SUBAPPLICATION Uebung_006_SAFE_AX_02 (* Wie Uebung_006_SAFE_AX, aber mit SF_EmergencyStop statt StartPermit/StartGate *)
  (* Standard: 61499-2; Description: Copyright (c) 2026 Meisterschulen am Ostbahnhof This program and the accompanying materials are made available under the terms of the Eclipse Public License 2.0 which is available at https://www.eclipse.org/legal/epl-2.0/ SPDX-License-Identifier: EPL-2.0 *)
  (* Version 1.0, 2026-10-09, Franz Höpfinger, Meisterschulen am Ostbahnhof, Zweite SAFE-Variante von Uebung_006_AX, diesmal mit dem PLCopen-Standardbaustein SF_EmergencyStop (Part 1 Ch. 6.5) statt der handgebauten StartPermit(E_RS)/StartGate(E_PERMIT)-Loesung aus Uebung_006_SAFE_AX. SF_EmergencyStop und SF_ResetButton sind im eingebetteten Muster (Figure 13 der Spec) ueber ResetRequest/ResetRequested verkoppelt: EmergencyStop fordert ResetButton nur dann zur Ueberwachung an, wenn tatsaechlich ein Reset noetig ist. S_StartReset=FALSE und S_AutoReset=FALSE: kein automatischer Wiederanlauf, RESET (I7) ist immer zwingend erforderlich. *)
  PACKAGE Uebungen;
  IMPORT logiBUS::io::DI::logiBUS_DI::Input_I1;
  IMPORT logiBUS::io::DI::logiBUS_DI::Input_I2;
  IMPORT logiBUS::io::DI::logiBUS_DI::Input_I7;
  IMPORT logiBUS::io::DI::logiBUS_DI::Input_I8;
  IMPORT logiBUS::io::DI::logiBUS_DI_Events::BUTTON_SINGLE_CLICK;
  IMPORT logiBUS::io::DQ::logiBUS_DO::Output_Q1;
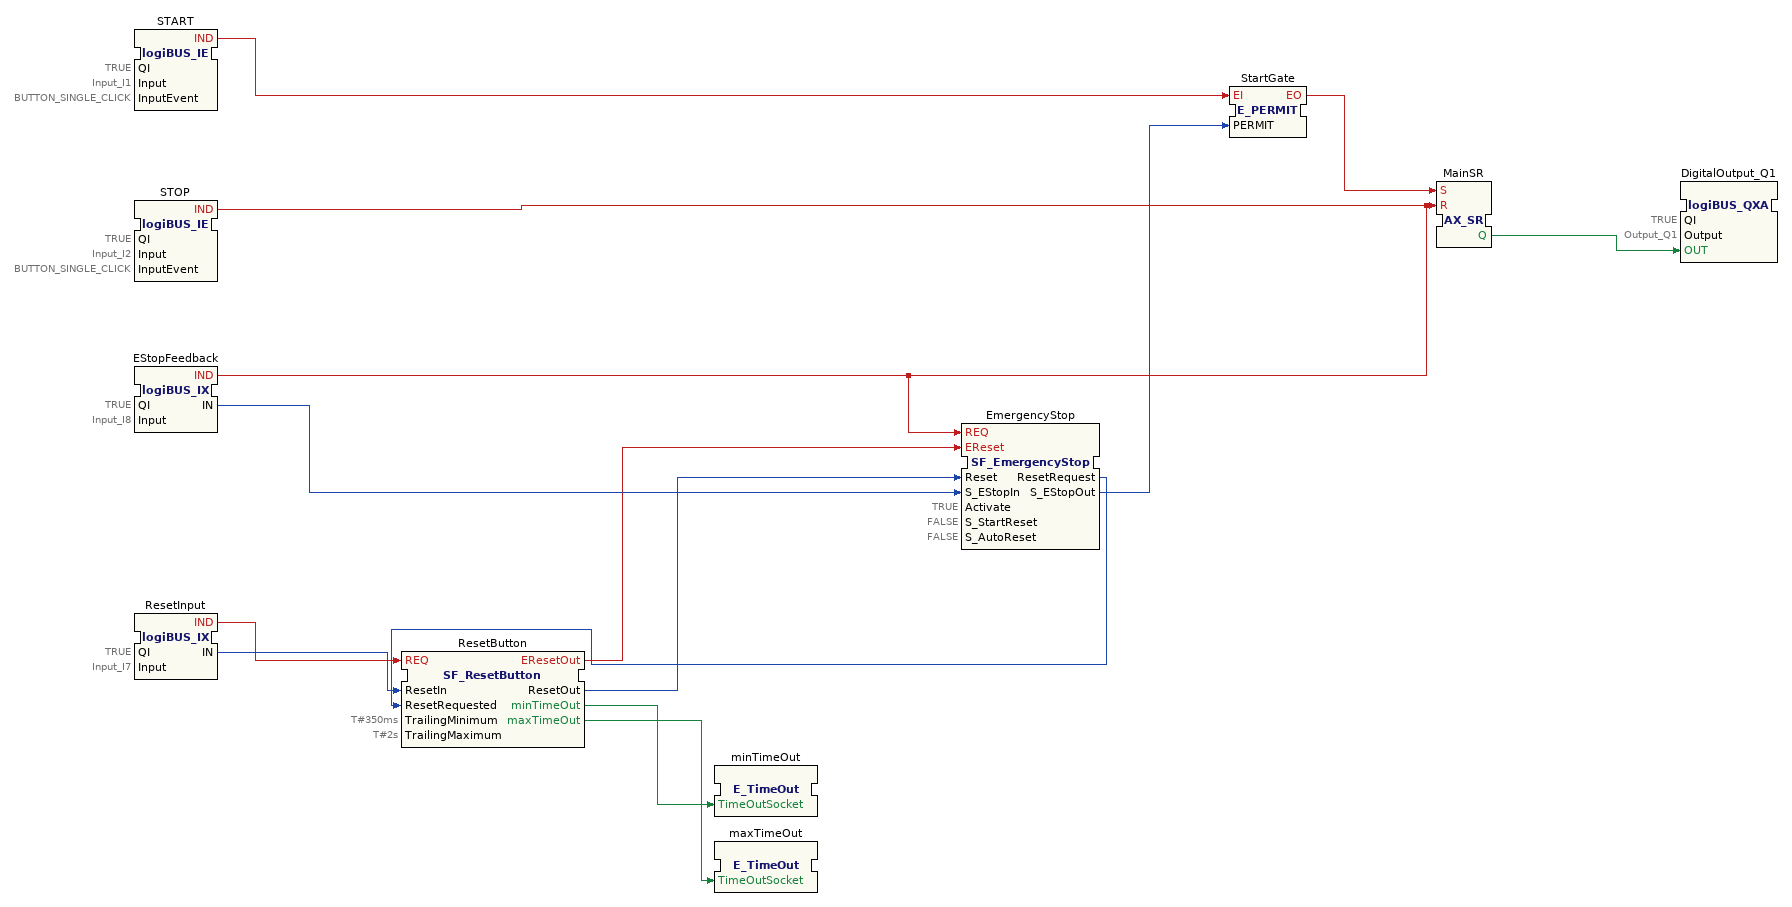
  FBS
    START : logiBUS::io::DI::logiBUS_IE(QI := TRUE, Input := Input_I1, InputEvent := BUTTON_SINGLE_CLICK); (* Taster START *)
    STOP : logiBUS::io::DI::logiBUS_IE(QI := TRUE, Input := Input_I2, InputEvent := BUTTON_SINGLE_CLICK); (* Hand-Stopp (nicht HW-Not-Halt) *)
    EStopFeedback : logiBUS::io::DI::logiBUS_IX(QI := TRUE, Input := Input_I8); (* I8=TRUE: Not-Halt-Kreis ok. I8=FALSE: Stop erkannt *)
    ResetInput : logiBUS::io::DI::logiBUS_IX(QI := TRUE, Input := Input_I7); (* Pegel+Event fuer SF_ResetButton *)
    ResetButton : logiBUS::safety::PLCopen::SF_ResetButton(TrailingMinimum := T#350ms, TrailingMaximum := T#2s);
    EmergencyStop : logiBUS::safety::PLCopen::SF_EmergencyStop(Activate := TRUE, S_StartReset := FALSE, S_AutoReset := FALSE);
    StartGate : iec61499::events::E_PERMIT; (* Laesst START nur bei Freigabe durch *)
    MainSR : adapter::events::unidirectional::AX_SR;
    DigitalOutput_Q1 : logiBUS::io::DQ::logiBUS_QXA(QI := TRUE, Output := Output_Q1);
    minTimeOut : iec61499::events::E_TimeOut;
    maxTimeOut : iec61499::events::E_TimeOut;
  END_FBS
  EVENT_CONNECTIONS
    START.IND TO StartGate.EI;
    StartGate.EO TO MainSR.S;
    STOP.IND TO MainSR.R;
    EStopFeedback.IND TO MainSR.R;
    EStopFeedback.IND TO EmergencyStop.REQ;
    ResetInput.IND TO ResetButton.REQ;
    ResetButton.EResetOut TO EmergencyStop.EReset;
  END_CONNECTIONS
  DATA_CONNECTIONS
    ResetInput.IN TO ResetButton.ResetIn;
    ResetButton.ResetOut TO EmergencyStop.Reset;
    EmergencyStop.ResetRequest TO ResetButton.ResetRequested;
    EStopFeedback.IN TO EmergencyStop.S_EStopIn;
    EmergencyStop.S_EStopOut TO StartGate.PERMIT;
  END_CONNECTIONS
  ADAPTER_CONNECTIONS
    MainSR.Q TO DigitalOutput_Q1.OUT;
    ResetButton.minTimeOut TO minTimeOut.TimeOutSocket;
    ResetButton.maxTimeOut TO maxTimeOut.TimeOutSocket;
  END_CONNECTIONS
END_SUBAPPLICATION
